# EPICS substitutions: example/exampleApp/Db/user.substitutions
# Example substitutions file

file "db/dbExample1.db" {
    { user = "xgc" }
}

file db/dbExample2.db {
    pattern { user, no, scan }
        { "xgc", 1, "1 second" }
        { "xgc", 2, "2 second" }
        { "xgc", 3, "5 second" }
}
